// TIA Portal V17 export
// export: Created 2025-03-07T09:24:24.5065681Z, ExportSetting WithDefaults, DisplayName Totally Integrated Automation Portal, DisplayVersion V17 Update 8, DisplayName TIA Portal Openness, DisplayVersion V17 Update 8, DisplayName TIA Portal Version Control Interface, DisplayVersion V17, DisplayName SINAMICS Startdrive Advanced, DisplayVersion V17 SP2, DisplayName SINAMICS Startdrive G110M, G120, G120C, G120D, G120P, G115D, DisplayVersion V17 SP2, DisplayName SINAMICS Startdrive G130, G150, S120, S150, SINAMICS MV, S210, DisplayVersion V17 SP2, DisplayName STEP 7 Professional, DisplayVersion V17 Update 8, DisplayName SINUMERIK ONE STEP 7 Toolbox, DisplayVersion V17 Update 12, DisplayName SINUMERIK 840D sl STEP 7 Toolbox, DisplayVersion V17 Update 12, DisplayName STEP 7 Safety, DisplayVersion V17 Update 6, DisplayName WinCC Advanced, DisplayVersion V17 Update 8
DATA_BLOCK "DB22535_TEMPERATURE_JKT_LOWER_HOPPER_2_UNIT_02"   // DB22535
{ DB_Accessible_From_OPC_UA := 'FALSE' }
VERSION : 0.1
// stored: AutoNumber false, DBAccessibleFromOPCUA false, DBAccessibleFromWebserver true, InstanceOfName FB22501_TEMPERATURE_JKT_CONTROL, InstanceOfType FB
"FB22501_TEMPERATURE_JKT_CONTROL"
   // VAR_INPUT
   //    iFEEDBACK_TEMP : Real;
   //    iCONTROL_ON_DELAYED : Bool;
   //    iBREAKER : Bool;
   //    iMANUAL_START_REQUEST : Bool;
   //    iMANUAL_STOP_REQUEST : Bool;
   // END_VAR
   // VAR_OUTPUT
   //    oANALOG_TEMP_VALUE : Int;
   //    oSwitchoncondition_on : Bool;
   // END_VAR
   // VAR
   //    DATA : Struct
   //       Start : Bool;
   //       Conditions : Bool;
   //       "Auto Cons." : Real;
   //       Consignment : Real;
   //       Min_Range : Real;
   //       Max_Range : Real;
   //       Lim_Lo : Real;
   //       Lim_HI : Real;
   //       "HMI Manual Cons." : Real;
   //       "HMI Feedback Value" : Real;
   //       "HMI Consignment" : Real;
   //    END_STRUCT;
   // END_VAR
BEGIN
END_DATA_BLOCK
